{attribute 'qualified_only'}
VAR_GLOBAL	
B1	AT %I* :BOOL;   	// 	Position Flasche
F1	AT %I* :BOOL;   	// 	Motorschutzschalter
S1	AT %I* :BOOL;   	// 	Taster Start
S2	AT %I* :BOOL;   	// 	Taster Stop
S3	AT %I* :BOOL;   	// 	Taster Vereinzelung
S4	AT %I* :BOOL;   	// 	Taster Quittieren
END_VAR

(* stored: Version 1.1.0.1, ProductVersion 3.1.4024.5
   GVL DI: Id {c2d05302-d374-4f85-80dd-41006a3e3277} *)
